// TIA Portal project "TimersUsingHMI" (V17)

(* hardware
DEVICE "HMI_1"  KTP700 Basic PN
   slot 0: "HMI_1"  KTP700 Basic PN  6AV2 123-2GB03-0AX0  17.0.0.0
   slot 1: "HMI_RT_1"  KTP700 Basic PN  6AV2 123-2GB03-0AX0  17.0.0.0
   slot 5: "HMI_1.IE_CP_1"  PROFINET Interface  17.0.0.0
      slot 1: "PROFINET Interface_1"  PROFINET Interface
         slot 1: "Port_1"  Port
DEVICE "S7-1200 station_1"  S7-1200 Station
   slot 0: "Rack_0"  S7-1200 Rack  Rack  V1.0
   slot 1: "PLC_1"  CPU 1214C DC/DC/DC  6ES7 214-1AG40-0XB0  V4.5
*)

// ===== PLC "PLC_1"  CPU 1214C DC/DC/DC =====

VAR_GLOBAL   // PLC tag table "Default tag table"
   "startPB" AT %I0.0 : Bool;
   "motor" AT %Q0.0 : Bool;
END_VAR

DATA_BLOCK "timerONDataBlock"   // DB2
{ S7_Optimized_Access := 'TRUE' }
VERSION : 0.1
   VAR
      elapsedTime : Time;
   END_VAR
BEGIN
END_DATA_BLOCK

// folder: System blocks/Program resources

DATA_BLOCK "timerON"   // DB1
{ S7_Optimized_Access := 'TRUE' }
AUTHOR : Simatic
FAMILY : IEC
NAME : IEC_TMR
VERSION : 1.0
// stored: InstanceOfName IEC_TIMER
"IEC_TIMER"
BEGIN
END_DATA_BLOCK

// folder: (top level)

ORGANIZATION_BLOCK "Main"   // OB1, LAD, ProgramCycle
TITLE = "Main Program Sweep (Cycle)"
{ S7_Optimized_Access := 'TRUE' }
VERSION : 0.1
   VAR_INPUT
      Initial_Call : Bool;   // Initial call of this OB
      Remanence : Bool;   // =True, if remanent data are available
   END_VAR
BEGIN

REGION Network 1
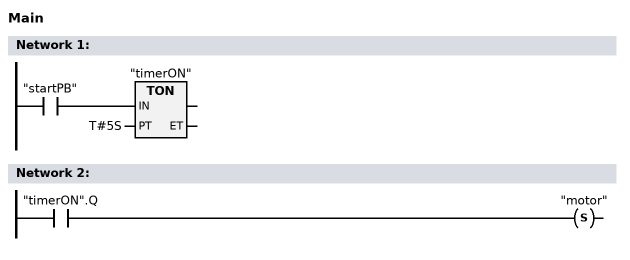
   "timerON".TON(IN := "startPB", PT := T#5S);
END_REGION

REGION Network 2
   RUNG wire#powerrail
      Contact( "timerON".Q )
      S_Coil( "motor" )
   END_RUNG
   // the same network as SCL:
   IF "timerON".Q THEN "motor" := TRUE; END_IF;
END_REGION
END_ORGANIZATION_BLOCK

(* ===== HMI "HMI_RT_1" =====
system functions are stored by id; their names below are inferred from use
connection "HMI_Connection_1": ETHERNET, SMART_S7_1200_OMS

HMI tags "Default tag table"
   "Tag_ScreenNumber" : UInt, internal
   "startPB" : Bool = PLC startPB AT %I0.0, 1 s
   "motor" : Bool = PLC motor AT %Q0.0, 1 s
   "timerONDataBlock_elapsedTime" : Time = PLC timerONDataBlock.elapsedTime, 1 s

Template "Template_1" 800x480
   Button "Exit" at 714,429 size 71x50; TextOff 'Exit'; PictureOff "ExitRuntime_KTP700_Basic_PN_TR"; PictureOn "ExitRuntime_KTP700_Basic_PN_TR"
      on Release: StopRuntime(0)
   Button "Template_Button" at 614,429 size 71x50; TextOff 'Text'
   Button "Template_Button_1" at 514,429 size 71x50; TextOff 'Text'
   Button "Template_Button_2" at 414,429 size 71x50; TextOff 'Text'
   Button "Language" at 314,429 size 71x50; TextOff 'Language'; PictureOff "ToggleLanguage_KTP700_Basic_PN_TR"; PictureOn "ToggleLanguage_KTP700_Basic_PN_TR"
      on Release: function_fb9197e8(-1)
   Button "Log on" at 214,429 size 71x50; TextOff 'Log on'; PictureOff "Login_KTP700_Basic_PN_TR"; PictureOn "Login_KTP700_Basic_PN_TR"
      on Release: function_a2a04561()
   Button "Alarms" at 114,429 size 71x50; TextOff 'Alarms'; PictureOff "AlarmDisplay_KTP700_Basic_PN_TR"; PictureOn "AlarmDisplay_KTP700_Basic_PN_TR"
      on Release: function_ef3f5d25("Alarm window_Unacknowledged", -1)
   Button "Start screen" at 14,429 size 71x50; TextOff 'Start screen'; PictureOff "NavigateHome_KTP700_Basic_PN_TR"; PictureOn "NavigateHome_KTP700_Basic_PN_TR"
      on Release: ActivateScreen("Root screen", 0)
   SymbolicIOField "Symbolic_IO_Field_Screen" at 2,9 size 691x33; TextOff '0'; TextOn '1'; TextList "TextList_ScreenNames"
      ProcessValue <- "Tag_ScreenNumber"
      on Change: ActivateScreenByNumber("Tag_ScreenNumber", 0)
   DateTimeField "HmiScreenItemData" at 695,25 size 105x25
   DateTimeField "HmiScreenItemData_1" at 695,0 size 105x25

screen "Root screen" 800x480, template "Template_1"
   on GenerateScreen: SetTag("Tag_ScreenNumber", 1)
   TextField "HmiScreenItemData_2" at 80,225 size 640x25; Text 'Welcome to our HMI platform. This is the main screen.'
   Button "HmiScreenItemData" at 36,87 size 159x47; TextOff 'Screen0'; PictureOff "Navigates to Screen0 for KTP700 Basic+ PN 17.0.0.0"; PictureOn "Navigates to Screen0 for KTP700 Basic+ PN 17.0.0.0"
      on Release: ActivateScreen("Screen0", 0)
   Button "HmiScreenItemData_1" at 36,146 size 159x47; TextOff 'Screen1'; PictureOff "Navigates to Screen1 for KTP700 Basic+ PN 17.0.0.0"; PictureOn "Navigates to Screen1 for KTP700 Basic+ PN 17.0.0.0"
      on Release: ActivateScreen("Screen1", 0)

screen "Screen0" 800x480, template "Template_1"
   on GenerateScreen: SetTag("Tag_ScreenNumber", 2)
   Button "Back" at 1,52 size 159x47; TextOff 'Back'
      on Release: ActivateScreen("Root screen", 0)
   Button "Button_1" at 266,133 size 96x32; TextOff 'Start'
      on Click: SetBit("startPB")
   Circle "Circle_1" at 288,239 size 48x48
      Visibility <- "motor"
      Appearance <- "motor"
   TextField "Text field_1" at 280,210 size 58x23; Text 'Motor'
   IOField "I/O field_1" at 523,162 size 96x32; FormatPattern 999
      ProcessValue <- "timerONDataBlock_elapsedTime"
   TextField "Text field_2" at 209,14 size 98x23; Text 'TON screen'

screen "Screen1" 800x480, template "Template_1"
   on GenerateScreen: SetTag("Tag_ScreenNumber", 3)
   TextField "HmiScreenItemData" at 80,225 size 640x25; Text 'Screen1'
   Button "Back" at 1,52 size 159x47; TextOff 'Back'
      on Release: ActivateScreen("Root screen", 0)
*)